(* IEC 61131-3 sources: fileTools/, 3 files *)

(* ---- fileTools.typ ---- *)
(********************************************************************
 * COPYRIGHT -- B&R Industrie-Elektronik GmbH
 ********************************************************************
 * Library: fileTools
 * Datei: fileTools.typ
 * Autor: wielando
 * Erstellt: 17. Juli 2012
 ********************************************************************
 * Datentypen der Library fileTools
 ********************************************************************)

TYPE

END_TYPE

(* ---- fileTools.fun ---- *)
(********************************************************************
 * COPYRIGHT -- B&R Industrie-Elektronik GmbH
 ********************************************************************
 * Library: fileTools
 * Datei: fileTools.fun
 * Autor: wielando
 * Erstellt: 17. Juli 2012
 ********************************************************************
 * Funktionen und Funktionsblöcke der Library fileTools
 ********************************************************************)

FUNCTION basename : UDINT (*Returns address to a string with the file name without path and extension*)
	VAR_INPUT
		pFileName : UDINT; (*File name*)
		pExtension : UDINT; (*File extension*)
	END_VAR
END_FUNCTION

FUNCTION getfileext : UINT (*Gets the file extension*)
	VAR_INPUT
		adrFileName : UDINT;
		adrExtention : UDINT;
	END_VAR
END_FUNCTION

FUNCTION hasExtension : BOOL
	VAR_INPUT
		pFilename : UDINT;
		pExtension : UDINT;
	END_VAR
END_FUNCTION

(* ---- fileTools.var ---- *)
(********************************************************************
 * COPYRIGHT -- B&R Industrie-Elektronik GmbH
 ********************************************************************
 * Library: fileTools
 * Datei: fileTools.var
 * Autor: wielando
 * Erstellt: 17. Juli 2012
 ********************************************************************
 * Konstanten der Library fileTools
 ********************************************************************)

VAR CONSTANT

END_VAR
